FUNCTION_BLOCK BaseProcess EXTENDS SM_BaseProcess (* default process *)
VAR_INPUT
	_state : INT; // internal state, may or may not be used
END_VAR
VAR_OUTPUT
END_VAR
VAR
END_VAR

// we make it easy for ourselves: every time the process is idle, we reset the startedStatus
IF statuses.busyStatus.idle THEN
	statuses.startedStatus(isStarted := FALSE);
END_IF

_update();

METHOD isIdle : BOOL
VAR_INPUT
END_VAR
isIdle := statuses.busyStatus.idle;
END_METHOD

METHOD _update
VAR_INPUT
END_VAR

IF actualStatus = '' THEN
    IF statuses.enabledStatus.disabled THEN
        actualStatus := '';
    ELSIF statuses.enabledStatus.enabled THEN
        IF statuses.healthStatus.good THEN
            IF statuses.busyStatus.busy THEN
                actualStatus := 'Busy';
            ELSIF statuses.busyStatus.idle THEN
                actualStatus := 'Idle';
            ELSE
                actualStatus := 'Good but UNKNOWN';
            END_IF
        ELSIF statuses.healthStatus.bad THEN
            IF statuses.busyStatus.busy THEN
                actualStatus := 'Error (busy)';
            ELSIF statuses.busyStatus.idle THEN
                actualStatus := 'Error';
            ELSE
                actualStatus := 'Bad but UNKNOWN';
            END_IF
        END_IF
    END_IF
END_IF

SUPER^();
END_METHOD

METHOD setBad
VAR_INPUT
END_VAR
statuses.healthStatus(isGood := FALSE);
END_METHOD

METHOD resetIfIdle
VAR_INPUT
END_VAR
IF statuses.busyStatus.idle  THEN
    
    statuses.healthStatus(isGood := TRUE, hasWarning := FALSE);
    setActualStatus('Idle');
    setFinished();
    
END_IF
END_METHOD

METHOD setBusy
VAR_INPUT
END_VAR
statuses.busyStatus(isBusy := TRUE);
END_METHOD

METHOD setFinished
VAR_INPUT
END_VAR
statuses.busyStatus(isBusy := FALSE);
statuses.startedStatus(isStarted := FALSE);
END_METHOD

METHOD setStarted
VAR_INPUT
END_VAR
statuses.startedStatus(isStarted := TRUE);
END_METHOD

METHOD isBusy : BOOL
VAR_INPUT
END_VAR
isBusy := statuses.busyStatus.busy;
END_METHOD

METHOD setActualStatus
VAR_INPUT
    msg : STRING;
END_VAR
actualStatus := msg;
END_METHOD

METHOD reset
VAR_INPUT
END_VAR
statuses.healthStatus(isGood := TRUE, hasWarning := FALSE);
statuses.busyStatus(isBusy := FALSE);
setActualStatus('Idle');
setFinished();
END_METHOD

METHOD setGood
VAR_INPUT
END_VAR
statuses.healthStatus(isGood := TRUE);
END_METHOD

METHOD isGood : BOOL
VAR_INPUT
END_VAR
isGood := statuses.healthStatus.good;
END_METHOD

METHOD FB_init : BOOL
VAR_INPUT
	bInitRetains : BOOL; // if TRUE, the retain variables are initialized (warm start / cold start)
	bInCopyCode : BOOL;  // if TRUE, the instance afterwards gets moved into the copy code (online change)
END_VAR
statuses.busyStatus(isBusy := FALSE);
statuses.startedStatus(isStarted := FALSE);
statuses.healthStatus(isGood := TRUE);
END_METHOD

METHOD isStarted : BOOL
VAR_INPUT
END_VAR
isStarted := statuses.startedStatus.started;
END_METHOD

END_FUNCTION_BLOCK

(* stored: Version 1.1.0.1, ProductVersion 3.1.4019.2
   POU BaseProcess: Id {e2ab5c41-31ef-48c8-b61a-d57074b4ff3e}, SpecialFunc None
   Method isIdle: Id {18d07c2c-58b4-4029-92b8-39a02fd85e95}
   Method _update: Id {1f2a76d0-b3bd-4061-861d-bc473f71fdc1}
   Method setBad: Id {4e820251-92ed-4334-82dd-5ee4c71a6c96}
   Method resetIfIdle: Id {500f85e4-9a9f-4942-9eb7-489cf50c14c3}
   Method setBusy: Id {66fc4e37-dbac-472c-af1b-eca343a03802}
   Method setFinished: Id {957dff39-b430-4be5-85a8-d6ce9b506983}
   Method setStarted: Id {96b5b580-871c-4d81-a317-6d80daeed38b}
   Method isBusy: Id {9f1fadd6-1bcf-4c39-a6df-a6ce5df8af37}
   Method setActualStatus: Id {af70697a-5f0b-40a9-8564-ac4be8c0aa57}
   Method reset: Id {b7caaf6d-f58e-442f-9122-5f4f83cda7fa}
   Method setGood: Id {c20e0cc3-4234-4706-bb57-b2ed40a729b8}
   Method isGood: Id {d46318a2-0ede-4d9b-9421-53fa21752ea0}
   Method FB_init: Id {d735d7c3-8cea-4285-bf52-ff51ef54a516}
   Method isStarted: Id {ff10beff-1a82-4137-81fe-85f8ffdac9d6} *)
